TYPE ST_ShiftCalendarV2 :
STRUCT
    SchemaVersion : UINT;
    UtcOffsetMin : DINT;
    Rows : ARRAY[1..PL_Fraktal.MAX_SHIFTS] OF ST_ShiftRowV2;
END_STRUCT
END_TYPE

(* stored: Version 1.1.0.1, ProductVersion 3.1.4024.12
   DUT ST_ShiftCalendarV2: Id {7317ae20-8098-47ca-91bd-77983b70f4fe} *)
